// TwinCAT 3 PLC project PlanarTrackMovement
// ProgramVersion: 3.1.4024.0
// libraries:
//   Tc2_Standard, * (Beckhoff Automation GmbH)
//   Tc2_System, * (Beckhoff Automation GmbH)
//   Tc2_Utilities, * (Beckhoff Automation GmbH)
//   Tc3_EventLogger, * (Beckhoff Automation GmbH)
//   Tc3_Mc3PlanarMotion, * (Beckhoff Automation GmbH)
//   Tc3_Module, * (Beckhoff Automation GmbH)
//   Tc3_Physics, * (Beckhoff Automation GmbH)
//   Tc3_XTS_Utility, * (Beckhoff Automation GmbH)
// project tree:
//   DUTs/ E_TrackNum.TcDUT (not stored), MoverSort.TcDUT (not stored)
//   / FB_XtsXlMoverUtility.TcPOU, PlcTask.TcTTO (not stored)
//   GVLs/ GVL_General.TcGVL, GVL_Mc3.TcGVL
//   POUs/ FB_PWM.TcPOU (not stored), Flashlight.TcPOU, ReadTcCom.TcPOU, FB_PlanarMover.TcPOU, MAIN.TcPOU, IsBetween.TcPOU (not stored)

// ---- GVLs/GVL_General.TcGVL
VAR_GLOBAL CONSTANT

	nNumMaxMovers : UDINT :=10;
	nNumMaxTracks : UDINT :=3;
 	fMagnetEntry : LREAL := 10000;//8750; //PLEASE ENTER THE MAGNET ENTRY!!!
	fMagnetExit : LREAL := 10900; //PLEASE ENTER THE MAGNET EXIT!!!
END_VAR

VAR_GLOBAL
	aStopPositions : ARRAY [1..nNumMaxMovers] OF LREAL := [2400, 1700, 1000, 300];
	XtsOutterLoopOid: OTCID := 16#1010480;	
	XtsShortcutOid: OTCID := 16#1010490;
	
	MoverArrive : BOOL;
	MoverArrived : BOOL;
END_VAR

VAR_GLOBAL PERSISTENT
	nNumMovers: UDINT := 4;
	nMoverSartupPos : ARRAY[1..nNumMaxMovers] OF MoverSort;
END_VAR

// ---- GVLs/GVL_Mc3.TcGVL


VAR_GLOBAL
	//Track_BigCircle		: 	MC_PlanarTrack; 	
	//Track_MainCircle	: 	MC_PlanarTrack;
 	//Track_SmallCircle	: 	MC_PlanarTrack;
	
	MC_Tracks    		:	ARRAY[1..3] OF MC_PlanarTrack;
	MC_Trackfeedback	:	ARRAY[1..3] OF MC_PlanarFeedback;
	TrackTrail 			:	MC_PlanarTrackTrail;
	


	fbPlanarMover		:	ARRAY[1..nNumMaxMovers] OF FB_PlanarMover;
	MoverFeedback		:	ARRAY[1..nNumMaxMovers] OF MC_PlanarFeedback;
	
	
	
	Mover				:	ARRAY[0..nNumMaxMovers] OF MoverSort;
	
		
	fbXtsXlMoverUtility :	ARRAY[1..nNumMaxMovers] OF FB_XtsXlMoverUtility;
END_VAR

// ---- POUs/FB_PlanarMover.TcPOU
FUNCTION_BLOCK FB_PlanarMover

VAR_INPUT
	nMoverId			: UDINT;
	iTcIoXtsXpuMover	: I_TcIoXtsXpuMover;
END_VAR

VAR
	_McPlanarMover	: MC_PlanarMover;
	_PlanarTrail    : MC_PlanarTrackTrail;
  	

END_VAR

PROPERTY IsCommandedInShortcut : BOOL
GET
VAR
	nCounter: UDINT := 0;
END_VAR
_mcPlanarMover.GetTrackTrailInformation(_PlanarTrail);

IF _PlanarTrail.Error OR _PlanarTrail.Size < 1 THEN
   IsCommandedInShortcut := FALSE;
   RETURN;
END_IF
   
FOR nCounter := 0 TO _PlanarTrail.Size - 1 DO
	IF _PlanarTrail.GetTrackOidAt(nCounter) = GVL_Mc3.MC_Tracks[E_Tracknum.Small].MCTOPLC_STD.TrackOID  THEN
		IsCommandedInShortcut := TRUE;
		RETURN;
	END_IF
END_FOR

IsCommandedInShortcut := FALSE;
END_GET
END_PROPERTY

METHOD JoinTrack

VAR_INPUT
	feedback: REFERENCE TO MC_PlanarFeedback;
END_VAR

VAR_IN_OUT
	track: MC_PlanarTrack;
END_VAR
_McPlanarMover.JoinTrack(feedback, track, 0, 0);
END_METHOD

PROPERTY McPlanarMover : REFERENCE TO MC_PlanarMover
GET
McPlanarMover ref= _McPlanarMover;
END_GET
END_PROPERTY

METHOD Update : PVOID
_mcPlanarMover.Update();


_mcPlanarMover.GetTrackTrailInformation(_PlanarTrail);

IF _PlanarTrail.Error OR _PlanarTrail.Size <= 1 THEN
   RETURN;
END_IF
   
//SmallCircle
IF _PlanarTrail.GetTrackOidAt(1) = MC_Tracks[E_TrackNum.Small].MCTOPLC_STD.TrackOID   THEN
	iTcIoXtsXpuMover.SetActiveTrackObjectId(XtsShortcutOid);
//BigCircle
ELSIF _PlanarTrail.GetTrackOidAt(1) =MC_Tracks[E_TrackNum.Big].MCTOPLC_STD.TrackOID THEN
	iTcIoXtsXpuMover.SetActiveTrackObjectId(XtsOutterLoopOid);
END_IF
END_METHOD

END_FUNCTION_BLOCK

// ---- FB_XtsXlMoverUtility.TcPOU
FUNCTION_BLOCK FB_XtsXlMoverUtility
VAR_INPUT
	EdtDriverOid: OTCID;
END_VAR

VAR_OUTPUT
	bBusy: BOOL;
	bDone: BOOL;
	bError: BOOL;
	bInit: BOOL;
	ipResultMessage: I_TcMessage := fbResult;
END_VAR

VAR
	fbResult: FB_TcMessage;
	_ipComObject: ITComObject;
	
	PID_TriggerLeave						: PTCID := 16#030802EF;
	PID_TriggerArrive						: PTCID := 16#030802EE;
	PID_IsVirtualFeedbackEnabled			: PTCID := 16#0308050B;
	PID_ConfiguredDetectionTrackObjectId	: PTCID := 16#030802F0;
	PID_StartupTrackPosition				: PTCID := 16#03080370;
END_VAR

IF NOT bInit THEN
	IF GetComObject(nObjectId:=EdtDriverOid) THEN
		bInit:=TRUE;
	END_IF
	RETURN;
END_IF

METHOD GetComObject : BOOL
VAR_INPUT
	nObjectId: OTCID;
END_VAR
IF FW_ObjMgr_GetObjectInstance(	oid		:= nObjectId, 
								iid		:= TC_GLOBAL_IID_LIST.IID_ITComObject, 
								pipUnk	:= ADR(_ipComObject)) = 0
THEN
	GetComObject := TRUE;
END_IF
END_METHOD

METHOD SetConfiguredDetectionTrackObjectId : BOOL
VAR_INPUT
	nConfiguredDetectionTrackObjectId: OTCID;
END_VAR

VAR
	nValue: OTCID;
	stEventEntry: TcEventEntry;
	pstEventEntry: REFERENCE TO TcEventEntry := stEventEntry;
END_VAR

VAR_INST
	hResult : HRESULT;
END_VAR
bError := FALSE;

nValue := nConfiguredDetectionTrackObjectId;

IF _ipComObject <> 0 THEN 
	 hResult := 	_ipComObject.TcSetObjPara(		pid := PID_ConfiguredDetectionTrackObjectId,
													nData := SIZEOF(nValue),
													pData := ADR(nValue),
													pgp := 0); 	
	IF hResult = 0 THEN
		SetConfiguredDetectionTrackObjectId := TRUE;
	ELSE
		HRESULTAdsErr_TO_TcEventEntry(hResult,stEventEntry);
		IF NOT fbResult.EqualsToEventEntryEx( stOther := stEventEntry) THEN
			fbResult.CreateEx(stEventEntry, 0);
			fbResult.Send(0);
			fbResult.Release();
		END_IF
		bError := TRUE;
	END_IF							
END_IF
END_METHOD

METHOD SetIsVirtualFeedbackEnabled : BOOL
VAR_INPUT
	bSetIsVirtualFeedbackEnabled: BOOL;
END_VAR

VAR
	nValue: BOOL;
	stEventEntry: TcEventEntry;
	pstEventEntry: REFERENCE TO TcEventEntry := stEventEntry;
END_VAR

VAR_INST
	hResult : HRESULT;
END_VAR
bError := FALSE;

nValue := bSetIsVirtualFeedbackEnabled;

IF _ipComObject <> 0 THEN 
	 hResult := 	_ipComObject.TcSetObjPara(		pid := PID_IsVirtualFeedbackEnabled,
													nData := SIZEOF(nValue),
													pData := ADR(nValue),
													pgp := 0); 	
	IF hResult = 0 THEN
		SetIsVirtualFeedbackEnabled := TRUE;
	ELSE
		HRESULTAdsErr_TO_TcEventEntry(hResult,stEventEntry);
		IF NOT fbResult.EqualsToEventEntryEx( stOther := stEventEntry) THEN
			fbResult.CreateEx(stEventEntry, 0);
			fbResult.Send(0);
			fbResult.Release();
		END_IF
		bError := TRUE;
	END_IF							
END_IF
END_METHOD

METHOD SetStartupTrackPosition : BOOL
VAR_INPUT
	nStartupTrackPosition: REAL;
END_VAR

VAR
	nValue: REAL;
	stEventEntry: TcEventEntry;
	pstEventEntry: REFERENCE TO TcEventEntry := stEventEntry;
END_VAR

VAR_INST
	hResult : HRESULT;
END_VAR
bError := FALSE;

nValue := nStartupTrackPosition;

IF _ipComObject <> 0 THEN 
	 hResult := 	_ipComObject.TcSetObjPara(		pid := PID_StartupTrackPosition,
													nData := SIZEOF(nValue),
													pData := ADR(nValue),
													pgp := 0); 	
	IF hResult = 0 THEN
		SetStartupTrackPosition := TRUE;
	ELSE
		HRESULTAdsErr_TO_TcEventEntry(hResult,stEventEntry);
		IF NOT fbResult.EqualsToEventEntryEx( stOther := stEventEntry) THEN
			fbResult.CreateEx(stEventEntry, 0);
			fbResult.Send(0);
			fbResult.Release();
		END_IF
		bError := TRUE;
	END_IF							
END_IF
END_METHOD

METHOD TriggerArrive : BOOL
VAR_INPUT
END_VAR

VAR
	nValue: BOOL;
	stEventEntry: TcEventEntry;
	pstEventEntry: REFERENCE TO TcEventEntry := stEventEntry;
END_VAR

VAR_INST
	hResult : HRESULT;
END_VAR
bError := FALSE;

nValue := TRUE;

IF _ipComObject <> 0 THEN 
	 hResult := 	_ipComObject.TcSetObjPara(		pid := PID_TriggerArrive,
													nData := SIZEOF(nValue),
													pData := ADR(nValue),
													pgp := 0); 	
	IF hResult = 0 THEN
		TriggerArrive := TRUE;
	ELSE
		HRESULTAdsErr_TO_TcEventEntry(hResult,stEventEntry);
		IF NOT fbResult.EqualsToEventEntryEx( stOther := stEventEntry) THEN
			fbResult.CreateEx(stEventEntry, 0);
			fbResult.Send(0);
			fbResult.Release();
		END_IF
		bError := TRUE;
	END_IF							
END_IF
END_METHOD

METHOD TriggerLeave : BOOL
VAR_INPUT
END_VAR

VAR
	nValue: BOOL;
	stEventEntry: TcEventEntry;
	pstEventEntry: REFERENCE TO TcEventEntry := stEventEntry;
END_VAR

VAR_INST
	hResult : HRESULT;
END_VAR
bError := FALSE;

nValue := TRUE;

IF _ipComObject <> 0 THEN 
	 hResult := 	_ipComObject.TcSetObjPara(		pid := PID_TriggerLeave,
													nData := SIZEOF(nValue),
													pData := ADR(nValue),
													pgp := 0); 	
	IF hResult = 0 THEN
		TriggerLeave := TRUE;
	ELSE
		HRESULTAdsErr_TO_TcEventEntry(hResult,stEventEntry);
		IF NOT fbResult.EqualsToEventEntryEx( stOther := stEventEntry) THEN
			fbResult.CreateEx(stEventEntry, 0);
			fbResult.Send(0);
			fbResult.Release();
		END_IF
		bError := TRUE;
	END_IF							
END_IF
END_METHOD

END_FUNCTION_BLOCK

// ---- POUs/Flashlight.TcPOU
FUNCTION_BLOCK Flashlight


VAR_INPUT
    Frequence:        REAL := 0.5;             (* Realwert: Frequenz in Hz *)
END_VAR
VAR_OUTPUT
    Error:            BOOL := FALSE;        (* Input Frequenz = 0 *)
    Blinker:            BOOL := FALSE;        (* Blinker *)
END_VAR
VAR
    Cyceltime:        TIME := T#0MS;

    TON_1:             TON;
    TON_2:             TON;
END_VAR


IF Frequence = 0 THEN
    Error := TRUE;
    Blinker := FALSE;
ELSE
    Error := FALSE;

    (* Aus Hz ms machen *)
    Cyceltime := LREAL_TO_TIME(( 1.0 / Frequence ) * 1000);

    TON_1(IN:= NOT TON_2.Q, PT:=Cyceltime , Q=>);

    TON_2(IN:= TON_1.Q , PT:=Cyceltime , Q=> );

    IF TON_1.Q = TRUE THEN
        Blinker := TRUE;
    ELSE
        Blinker := FALSE;
    END_IF;

END_IF;

END_FUNCTION_BLOCK

// ---- POUs/ReadTcCom.TcPOU
FUNCTION_BLOCK ReadTcCom
VAR_INPUT
	
END_VAR
VAR_OUTPUT
	bBusy 				: BOOL;
	bDone 				: BOOL;
	bError 				: BOOL;
	bGetComObject	: BOOL;
END_VAR
VAR
	
	_nObjectId				: OTCID;
	_ipComObject 			: ITComObject;
	_nSoftDriveOid			: OTCID;
	PID_Value	: PTCID := 	16#05030149;
END_VAR

METHOD GetComObject : BOOL
VAR_INPUT
	nObjectId	: OTCID;
END_VAR
IF FW_ObjMgr_GetObjectInstance(	oid		:= nObjectId, 
								iid		:= TC_GLOBAL_IID_LIST.IID_ITComObject, 
								pipUnk	:= ADR(_ipComObject)) = 0
THEN
	GetComObject := TRUE;
END_IF
END_METHOD

METHOD GetValue : ARRAY[1..nNumMovers] OF OTCID
VAR_INPUT
	PID_Value 		: otcid;
END_VAR
VAR
	Value			: ARRAY[1..nNumMovers] OF OTCID;
	nData 			: UDINT := SIZEOF(Value);
	pData 			: PVOID := ADR(Value);
	stEventEntry	: TcEventEntry;
	pstEventEntry	: REFERENCE TO TcEventEntry REF= stEventEntry;
	
END_VAR
VAR_INST
	hResult : HRESULT;
END_VAR
IF _ipComObject <> 0  THEN
	 hResult := _ipComObject.TcGetObjPara(
				pid 	:= PID_Value,
				nData 	:= nData,
				pData 	:= pData,
				pgp   	:=0) ;
	IF hResult = 0	THEN
		GetValue := Value;
		bError := FALSE;
	ELSE
		bError := TRUE;
	END_IF
END_IF
END_METHOD

END_FUNCTION_BLOCK

// ---- POUs/MAIN.TcPOU
PROGRAM MAIN
VAR
		
	bAllDone		: BOOL;
	bStopSequence	: BOOL;
	
	nCase 		: INT;
	nMoveState		: ARRAY[1..nNumMaxMovers] OF INT;
	
	aDynamics	: ARRAY[1..nNumMaxMovers] OF DynamicConstraint_PathXY;
	aMoveOnTrackOptions : ARRAY[1..20] OF ST_MoveOnTrackOptions;
	
	fbXtsEnvironment: FB_TcIoXtsEnvironment;
	
	nForCounter: UDINT;
	M,N,T,Tr,i : UDINT;
	dynamics: INT;
	
	// Magnet
	MagnetValue AT%Q*: INT;
	bMagnetOn : BOOL;	
	stPositionInfo: ST_PositionInfo;
		
	pwm: FB_PWM;
	
	IsMoverCommandedInShortcut: BOOL;
	IsMoverInBlockingArea: BOOL;
	nActStopPos: UINT := 1;
	Fp_error : R_Trig;
	Velo : LREAL := 500;
	Velom1 : LREAL := 500;
	Switch : BOOL;
	WithoutSwitch : BOOL;
	SwtichOnly: BOOL;
	
	MoverStop 		AT%I* : BOOL;
	MoverStopDone 	AT%Q* : BOOL;
	Info 			AT%Q* : BOOL;
	Operating		AT%Q* : BOOL;
	Process			AT%Q* : BOOL;
	Fault			AT%Q* : BOOL;
	Emergency		AT%Q* : BOOL;
	
	Voltage1 		AT%I* : UDINT;
	Voltage2 		AT%I* : UDINT;
	
	
	TcRestart : TC_Restart;
	Restart : BOOL;
	busy : BOOL;
	fp_start : R_Trig;
	bStartSequence: BOOL;
	
	FP_Counter : r_trig;
	Switchcounter : DINT;
	SwitchCurrent: INT :=12; 
	test : LREAL;
	Horntimer : tp; 
	R_trigHorn : R_trig;
	
	TestPowerMat : BOOL;
	StopPos : LREAL := 7611;
	StopTime : TIME := T#8S;
	StopTimer :ARRAY[1..nNumMaxMovers] OF ton;
	StartTimer :ARRAY[1..nNumMaxMovers] OF BOOL;
	
	
	MoverPos :ARRAY[1..nNumMaxMovers] OF PositionXYC;
	ArcLength :ARRAY[1..nNumMaxMovers] OF LREAL;
	TrackPos :ARRAY[1..nNumMaxMovers] OF ARRAY[1..nNumMaxTracks] OF PositionXYC;
	fbFlashlight : Flashlight;
END_VAR

fbXtsEnvironment.Init(TRUE);

Emergency := NOT  MoverStop;


R_trigHorn(clk := MoverStop);
Horntimer(in:= ( R_trigHorn.Q ) , PT:= T#5S,Q=> info);
fbFlashlight(Frequence:=5 , Error=> , Blinker=> );

IF  NOT Horntimer.Q AND MoverStop THEN
	Process := TRUE;
ELSIF Horntimer.Q THEN
	Process:= fbFlashlight.Blinker;
	
ELSE	
	Process := FALSE;
END_IF






IF NOT fbXtsEnvironment.P_IsInitialized THEN
	RETURN;
END_IF

fbXtsEnvironment.XpuTcIo(1).GetPartOids();
IF NOT MoverArrived AND nMoverSartupPos[1].MoverPos <> 0 AND FALSE THEN
	FOR i := 1 TO nNumMaxMovers DO
		fbXtsXlMoverUtility[i].SetConfiguredDetectionTrackObjectId(  nMoverSartupPos[i].TrackID );		
		fbXtsXlMoverUtility[i].SetStartupTrackPosition( (nMoverSartupPos[i].MoverPos)) ;
		fbXtsXlMoverUtility[i].TriggerArrive();
		MoverArrived := TRUE;
	END_FOR	
END_IF



IF NOT MoverStop AND NOT MoverStopDone THEN
	FOR nForCounter:=1 TO nNumMovers DO
		aDynamics[nForCounter].SetValuesVADJ(4000, 4000, 4000, 15000);
		nCase := 140;
		//fbPlanarMover[nForCounter].McPlanarMover.Halt(MoverFeedback[nForCounter], aDynamics[nForCounter]);
	END_FOR		

ELSIF 	MoverStop THEN
	MoverStopDone := FALSE;
END_IF


	TcRestart(
	NETID:= '', 
	RESTART:= Restart, 
	TMOUT:=T#5S , 
	BUSY=>busy , 
	ERR=> , 
	ERRID=> );


fp_start(clk:=bStartSequence);
IF fp_start.Q THEN
	nCase := 10;
	bStartSequence := FALSE;
END_IF


IsMoverCommandedInShortcut := FALSE;
IsMoverInBlockingArea := FALSE;
FOR M := 1 TO nNumMovers DO///Movers
	StopTimer[M](in:=StartTimer[m],PT:=StopTime);
	fbPlanarMover[m].nMoverId := nForCounter;
	fbPlanarMover[m].iTcIoXtsXpuMover := fbXtsEnvironment.XpuTcIo(1).MoverTcIo(TO_UINT(m));
	fbPlanarMover[m].Update();
	
	GVL_mc3.Mover[M].MoverPos :=test :=fbPlanarMover[M].McPlanarMover.MCTOPLC.SETONTRACK.SetPos;
	GVL_mc3.Mover[M].TrackID:= fbPlanarMover[M].McPlanarMover.MCTOPLC.SETONTRACK.TrackOID;
	GVL_mc3.Mover[M].MoverNumber := M;
	
	MoverPos[M].SetValuesXYC(fbPlanarMover[M].McPlanarMover.MCTOPLC.SET.SetPos.x ,fbPlanarMover[M].McPlanarMover.MCTOPLC.SET.SetPos.y,fbPlanarMover[M].McPlanarMover.MCTOPLC.SET.SetPos.c);
	
	TR := Tr+1;
	IF Tr >= nNumMaxTracks THEN
		Tr :=1;
	END_IF
	ArcLength[M] :=GVL_Mc3.MC_Tracks[Tr].GetArcLengthClosestTo(MoverPos[M]);
	GVL_Mc3.MC_Tracks[Tr].GetPositionAt(ArcLength[M],TrackPos[M][Tr]);
	
	IF ABS(MoverPos[m].x - TrackPos[M][Tr].x) < 1 AND  ABS(MoverPos[m].y - TrackPos[M][Tr].y) < 1 THEN
 		GVL_mc3.Mover[M].MoverTrackNr := Tr;
	END_IF	
	
	
		
	IsMoverCommandedInShortcut := IsMoverCommandedInShortcut OR fbPlanarMover[M].IsCommandedInShortcut;
	IsMoverInBlockingArea := IsMoverInBlockingArea OR (Mover[M].TrackID = GVL_Mc3.MC_Tracks[E_TrackNum.main].MCTOPLC_STD.TrackOID AND IsBetween(Mover[M].MoverPos, fMagnetEntry - 100, fMagnetExit + 100));
	MoverFeedback[M].Update();
	
	Fp_error(clk := fbPlanarMover[M].McPlanarMover.Error AND ncase= 100);
	IF Fp_error.Q THEN
		nCase := 140;
		Fault := TRUE;
		bMagnetOn := FALSE;
	
	END_IF
END_FOR

FOR T := 1 TO nNumMaxTracks DO 
	MC_Tracks[T].Update();
	MC_Trackfeedback[T].Update();
	
END_FOR

CASE nCase OF
	10:
		FOR nForCounter := 1 TO fbXtsEnvironment.XpuTcIo(1).GetPartCount() DO
			fbXtsEnvironment.XpuTcIo(1).PartTcIo(TO_UINT(nForCounter)).TriggerReset();
		END_FOR
		Fault := FALSE;
		nCase := 20;

	20:
		FOR T := 1 TO nNumMaxTracks DO 
			MC_Tracks[T].Enable(MC_Trackfeedback[T]);
		END_FOR
				nCase := 30;
		
		
	30: 
		IF MC_Trackfeedback[1].Done AND MC_Trackfeedback[2].Done AND MC_Trackfeedback[3].Done THEN
			nCase := 35;
		END_IF
		
		
	35:
		FOR nForCounter:=1 TO nNumMovers DO
			fbPlanarMover[nForCounter].McPlanarMover.Reset(MoverFeedback[nForCounter]);
		END_FOR
		nCase := 36;	
		
		
	36:	
		bAllDone:=TRUE;
		FOR nForCounter:=1 TO nNumMovers DO
			bAllDone:=bAllDone AND MoverFeedback[nForCounter].Done;
		END_FOR
		
		IF bAllDone THEN
			nCase := 40;
		END_IF
		
		
	40:
		FOR nForCounter:=1 TO nNumMovers DO
			fbPlanarMover[nForCounter].McPlanarMover.Enable(MoverFeedback[nForCounter]);
		END_FOR
		nCase := 50;
	
		
	50:
		bAllDone:=TRUE;
		FOR nForCounter:=1 TO nNumMovers DO
			bAllDone:=bAllDone AND MoverFeedback[nForCounter].Done;
		END_FOR
		
		IF bAllDone THEN
			nCase := 60;
		END_IF

	//55:

	60:
		FOR nForCounter:=nNumMovers TO 1  BY -1 DO
			fbPlanarMover[nForCounter].JoinTrack(MoverFeedback[nForCounter], GVL_Mc3.MC_Tracks[3]);//  Mover[nForCounter].MoverTrackNr]);//
		END_FOR
		
		nCase := 70;
		
		
	70:
		bAllDone:=TRUE;
		FOR nForCounter:=1 TO nNumMovers DO
			bAllDone:=bAllDone AND MoverFeedback[nForCounter].Done;
		END_FOR
		
		IF bAllDone THEN
			nCase := 80;
		END_IF
		
	80:	
		FOR nForCounter:=1 TO nNumMovers DO
			nMoveState[nForCounter] := 0;
			aMoveOnTrackOptions[nForCounter].direction := MC_Direction.mcDirectionPositive;
			aMoveOnTrackOptions[nForCounter].gapMode := MC_GAP_MODE_ON_TRACK.Fast1D;
		END_FOR
		
		nCase := 90;

	100:
		
		FOR nForCounter:=1 TO nNumMovers DO
			aDynamics[nForCounter].SetValuesVADJ(Velo, 4000, 4000, 10000); // (Velo+100, 4000, 4000, 10000); add velo 100 to make a platoon 
			aMoveOnTrackOptions[nForCounter].gap:= 1500; //900 // gap 900 to make a platoon //1500 or 2300 for switches
		END_FOR
	aDynamics[1].SetValuesVADJ(Velo-Velom1, 4000, 4000, 10000);
		FOR nForCounter:=1 TO nNumMovers DO
			CASE nMoveState[nForCounter] OF
				
				0: // Track 3 Main Cycel 
					fbPlanarMover[nForCounter].McPlanarMover.MoveOnTrack(MoverFeedback[nForCounter], GVL_Mc3.MC_Tracks[E_TrackNum.Main],  GVL_Mc3.MC_Tracks[E_TrackNum.Main].GetLength()-1000, aDynamics[nForCounter], aMoveOnTrackOptions[nForCounter]);
					nMoveState[nForCounter] := 10;
					
				10:
					IF Mover[nForCounter].MoverPos > GVL_Mc3.MC_Tracks[E_TrackNum.Main].GetLength()-4000  AND  Mover[nForCounter].TrackID =   GVL_Mc3.MC_Tracks[E_TrackNum.Main].MCTOPLC_STD.TrackOID    THEN//     MCTrackOid_MainSemicircle THEN
						IF (NOT Switch  AND  NOT SwtichOnly) OR WithoutSwitch OR IsMoverCommandedInShortcut THEN
							nMoveState[nForCounter] := 20; // 20 - BigCycel
							IF NOT  WithoutSwitch THEN
								Switch := TRUE;
							ELSE	
								Switch := FALSE;
							END_IF
						ELSE
							nMoveState[nForCounter] := 40;  // 40- SmallCycel
							IsMoverCommandedInShortcut := TRUE;
							Switch := FALSE;
						END_IF
					END_IF

				
				20:
					fbPlanarMover[nForCounter].McPlanarMover.MoveOnTrack(MoverFeedback[nForCounter], GVL_Mc3.MC_Tracks[E_TrackNum.Big], GVL_Mc3.MC_Tracks[E_TrackNum.Big].GetLength()-1000, aDynamics[nForCounter],aMoveOnTrackOptions[nForCounter]);
					nMoveState[nForCounter] := 30;
				
					
				30:
					IF Mover[nForCounter].MoverPos > GVL_Mc3.MC_Tracks[E_TrackNum.Big].GetLength()-4000 AND  Mover[nForCounter].TrackID = GVL_Mc3.MC_Tracks[E_TrackNum.Big].MCTOPLC_STD.TrackOID    THEN//      MCTrackOid_BigSemicircle THEN
						nMoveState[nForCounter] := 60;
					END_IF				
				
			
				40:
					fbPlanarMover[nForCounter].McPlanarMover.MoveOnTrack(MoverFeedback[nForCounter], GVL_Mc3.MC_Tracks[E_TrackNum.Small], (GVL_Mc3.MC_Tracks[E_TrackNum.Small].GetLength()/2), aDynamics[nForCounter], aMoveOnTrackOptions[nForCounter]);
					nMoveState[nForCounter] := 45;	

				45:
					IF MoverFeedback[nForCounter].Done THEN
						fbPlanarMover[nForCounter].McPlanarMover.MoveOnTrack(MoverFeedback[nForCounter], GVL_Mc3.MC_Tracks[E_TrackNum.Small], GVL_Mc3.MC_Tracks[E_TrackNum.Small].GetLength()-1000, aDynamics[nForCounter], aMoveOnTrackOptions[nForCounter]);
						nMoveState[nForCounter] := 50;
					END_IF

			
				50:
					IF Mover[nForCounter].MoverPos > GVL_Mc3.MC_Tracks[E_TrackNum.small].GetLength()-4000 AND  Mover[nForCounter].TrackID = GVL_Mc3.MC_Tracks[E_TrackNum.Small].MCTOPLC_STD.TrackOID    THEN// MCTrackOid_Shortcut THEN
						nMoveState[nForCounter] := 60;
					END_IF
					
				60:
					IF  TestPowerMat  THEN
						nMoveState[nForCounter] := 70;
					ELSE
						nMoveState[nForCounter] := 0;	
					END_IF
				70:
					fbPlanarMover[nForCounter].McPlanarMover.MoveOnTrack(MoverFeedback[nForCounter], GVL_Mc3.MC_Tracks[E_TrackNum.Main], StopPos, aDynamics[nForCounter], aMoveOnTrackOptions[nForCounter]);
					nMoveState[nForCounter] := 80;
				80:
					IF MoverFeedback[nForCounter].Done THEN
						StartTimer[nForCounter] := TRUE;
						nMoveState[nForCounter] := 85;
					END_IF
				85:
					IF 	StopTimer[nForCounter].Q THEN
						StartTimer[nForCounter] := FALSE;
						nMoveState[nForCounter] := 0;	
					END_IF
				END_CASE
		
		END_FOR

		IF bStopSequence AND NOT(IsMoverInBlockingArea) THEN
			nCase := 110;
			bStopSequence := FALSE;
		END_IF
		110:
			N:= nNumMovers;
			FOR nForCounter:=1 TO nNumMovers DO		
				GVL_General.aStopPositions[nForCounter] := TO_LREAL(  fbXtsEnvironment.XpuTcIo(1).MoverTcIo(TO_UINT(N)).GetSimulatedStartUpPosition());
				N := N -1;
			END_FOR
			nCase := 120;
		
		120:	
			nActStopPos := UDINT_TO_UINT(nNumMaxMovers-nNumMovers+1);
			FOR nForCounter:=1 TO nNumMovers DO
				aDynamics[nForCounter].SetValuesVADJ(1000, 4000, 4000, 10000);
				nMoveState[nForCounter] := 0;
				fbPlanarMover[nForCounter].McPlanarMover.MoveOnTrack(MoverFeedback[nForCounter], GVL_Mc3.MC_Tracks[E_TrackNum.main], 300, aDynamics[nForCounter],aMoveOnTrackOptions[nForCounter]);
			END_FOR

			nCase:= 130; 
		130:
			FOR nForCounter:=1 TO nNumMaxMovers - (nNumMaxMovers -nNumMovers)  DO
				CASE nMoveState[nForCounter] OF
					0:								
						
						IF Mover[nForCounter].MoverPos < 300 AND  Mover[nForCounter].TrackID = GVL_Mc3.MC_Tracks[E_TrackNum.main].MCTOPLC_STD.TrackOID THEN
							aMoveOnTrackOptions[nForCounter].gap:= 700;
							fbPlanarMover[nForCounter].McPlanarMover.MoveOnTrack(MoverFeedback[nForCounter], GVL_Mc3.MC_Tracks[E_TrackNum.main], aStopPositions[nActStopPos], aDynamics[nForCounter], aMoveOnTrackOptions[nForCounter]);
							nActStopPos := nActStopPos + 1;
							nMoveState[nForCounter] := 10;
						END_IF
				END_CASE
			END_FOR
		
			bAllDone := TRUE;
			FOR nForCounter:=1 TO nNumMovers DO
				IF NOT(MoverFeedback[nForCounter].Done OR MoverFeedback[nForCounter].Error) THEN
					bAllDone := FALSE;
					EXIT;
				END_IF
			END_FOR
			
			IF bAllDone THEN
				nCase := 150;
			END_IF
		
		140:
			FOR nForCounter:=1 TO nNumMovers DO
				fbPlanarMover[nForCounter].McPlanarMover.Halt(MoverFeedback[nForCounter], aDynamics[nForCounter]);
			END_FOR	
			
			nCase := 145;
			
		145:
			bAllDone := TRUE;
			FOR nForCounter:=1 TO nNumMovers DO
				IF NOT(MoverFeedback[nForCounter].Done OR MoverFeedback[nForCounter].Error) THEN
					bAllDone := FALSE;
					EXIT;
				END_IF
			END_FOR
			
			IF bAllDone THEN
				nCase := 150;
			END_IF
		
		//Disable
		150:
			MoverStopDone := TRUE;
			FOR nForCounter:=1 TO nNumMovers DO
				fbPlanarMover[nForCounter].McPlanarMover.Disable(MoverFeedback[nForCounter]);
			END_FOR
				
			nCase := 0;
END_CASE

bMagnetOn := FALSE;
FOR nForCounter:=1 TO nNumMovers DO
	stPositionInfo := fbXtsEnvironment.XpuTcIo(1).MoverTcIo(TO_UINT(nForCounter)).GetPositionInfo();
	IF stPositionInfo.nTrackObjectId = XtsShortcutOid AND (IsBetween(stPositionInfo.fTrackPosition, fMagnetEntry - (Velo*0.1), fMagnetExit))  THEN
		bMagnetOn := TRUE;
	END_IF
END_FOR

pwm();
	
IF bMagnetOn AND NOT Fault  AND   MoverStop THEN
//Rob July 3 Magnets rescaled 	MagnetValue := SwitchCurrent*1310;
	MagnetValue := SwitchCurrent*2047;  //july 3 scaling, 10V = 16A 
ELSE
 	MagnetValue := 0;
END_IF

FP_Counter(clk:=bMagnetOn);

IF FP_Counter.Q THEN
	Switchcounter := Switchcounter+1;

END_IF

END_PROGRAM
